ADAPTER L3_APart
  (* Standard: 61499-1 *)
  (* Version 0.0, 2008-04-22, EQUEROL, UJI *)
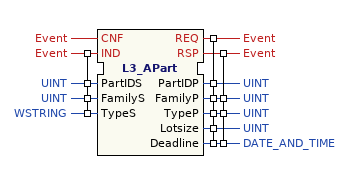
  EVENT_INPUT
    CNF; (* Confirmation to the socket *)
    IND WITH TypeS, FamilyS, PartIDS; (* Indication to the socket *)
  END_EVENT
  EVENT_OUTPUT
    REQ WITH PartIDP, FamilyP, TypeP, Lotsize, Deadline; (* Request from the plug *)
    RSP WITH Deadline, FamilyP, TypeP; (* Response from de plug *)
  END_EVENT
  VAR_INPUT
    PartIDS : UINT; (* Identifier of the last created part *)
    FamilyS : UINT; (* Part's Family *)
    TypeS : WSTRING; (* Part's Type *)
  END_VAR
  VAR_OUTPUT
    PartIDP : UINT; (* Identifier of the 1st part *)
    FamilyP : UINT; (* Part's Family *)
    TypeP : UINT; (* Part's type *)
    Lotsize : UINT; (* Number of parts to be manufactured *)
    Deadline : DATE_AND_TIME; (* Deadline of the next part to be delivered *)
  END_VAR
  SERVICE SOCKET/PLUG
    SEQUENCE request_confirm
      SOCKET.REQ(REQD) -> PLUG.REQ(REQD);
      PLUG.CNF(CNFD) -> SOCKET.CNF(CNFD);
    END_SEQUENCE
    SEQUENCE indication_response
      PLUG.IND(INDD) -> SOCKET.IND(INDD);
      SOCKET.RSP(RSPD) -> PLUG.RSP(RSPD);
    END_SEQUENCE
  END_SERVICE
END_ADAPTER
